// TIA Portal V17 export
// export: Created 2025-03-10T13:11:52.9134502Z, ExportSetting WithDefaults, DisplayName Totally Integrated Automation Portal, DisplayVersion V17 Update 8, DisplayName TIA Portal Openness, DisplayVersion V17 Update 8, DisplayName TIA Portal Version Control Interface, DisplayVersion V17, DisplayName SINAMICS Startdrive Advanced, DisplayVersion V17 SP2, DisplayName SINAMICS Startdrive G110M, G120, G120C, G120D, G120P, G115D, DisplayVersion V17 SP2, DisplayName SINAMICS Startdrive G130, G150, S120, S150, SINAMICS MV, S210, DisplayVersion V17 SP2, DisplayName STEP 7 Professional, DisplayVersion V17 Update 8, DisplayName SINUMERIK ONE STEP 7 Toolbox, DisplayVersion V17 Update 12, DisplayName SINUMERIK 840D sl STEP 7 Toolbox, DisplayVersion V17 Update 12, DisplayName STEP 7 Safety, DisplayVersion V17 Update 6, DisplayName WinCC Advanced, DisplayVersion V17 Update 8
TYPE "LBP_typeChanX"
TITLE = Channel interface / Interfaz de canal / Kanalschnittstelle
// User data type for blocks LBP_Chan1 [DB21] .. LBP_Chan10 [DB30] / Tipo de dato de usuario para bloques LBP_Chan1 [DB21] .. LBP_Chan10 [DB30] / Anwender-Datentyp für Bausteine LBP_Chan1 [DB21] .. LBP_Chan10 [DB30]
// stored: IsFailsafeCompliant false
   STRUCT
      f0_0 : Bool;
      f0_1 : Bool;
      f0_2 : Bool;
      A_DRF : Bool;   // DRF aktivieren / Activate DRF / Activar DRF
      A_SBL : Bool;   // Einzelsatz aktivieren / Activate single block / Activar secuencia individual
      A_M01 : Bool;   // M01 aktivieren / Activate M01 / Activar M01
      A_DRY : Bool;   // Probelauf Vorschub aktivieren / Activate dry run feedrate / Activar avance recorrido de prueba
      f0_7 : Bool;
      A_Ref : Bool;   // Referenzieren aktivieren / Activate referencing / Activar referenciado
      A_ProtZone : Bool;   // Schutzbereiche aktivieren / Enable protection zones / Activar zonas protegidas
      A_SynOff : Bool;   // Synchronaktion Aus / Synchronous action off / Acción síncrona desactivada
      A_TM_TimOut : Bool;   // Timeout aktivieren (TM) / Activate time-out (TM) / Activar timeout (TM)
      A_CLC_Stop : Bool;   // CLC Stopp / CLC stop / Parada CLC
      A_CLC_OR : Bool;   // CLC Override / CLC override / Corrección CLC
      A_PLC_ActCompl : Bool;   // PLC-Aktion abgeschlossen / PLC action completed / Acción PLC finalizada
      A_ProgTest : Bool;   // Programmtest aktivieren / Activate program test / Activar test de programa
      A_SKP0 : Bool;   // Ausblendsatz \0 aktivieren / Activate skip block \0 / Activar omisión de bloque \0
      A_SKP1 : Bool;   // Ausblendsatz \1 aktivieren / Activate skip block \1 / Activar omisión de bloque \1
      A_SKP2 : Bool;   // Ausblendsatz \2 aktivieren / Activate skip block \2 / Activar omisión de bloque \2
      A_SKP3 : Bool;   // Ausblendsatz \3 aktivieren / Activate skip block \3 / Activar omisión de bloque \3
      A_SKP4 : Bool;   // Ausblendsatz \4 aktivieren / Activate skip block \4 / Activar omisión de bloque \4
      A_SKP5 : Bool;   // Ausblendsatz \5 aktivieren / Activate skip block \5 / Activar omisión de bloque \5
      A_SKP6 : Bool;   // Ausblendsatz \6 aktivieren / Activate skip block \6 / Activar omisión de bloque \6
      A_SKP7 : Bool;   // Ausblendsatz \7 aktivieren / Activate skip block \7 / Activar omisión de bloque \7
      A_StrokEnab : Bool;   // Hub aktivieren / Stroke enable / Activar carrera
      A_ManStrokEnab : Bool;   // Manuelle Hub-Aktivierung / Manual stroke enable / Habilitación manual de carrera
      A_StrokSup : Bool;   // Hub-Unterdrückung / Stroke suppression / Supresión de carrera
      A_StrokDelayed : Bool;   // Hub verzögert / Stroke delayed / Carrera retardada
      A_StrokStop : Bool;   // Hub läuft nicht / Stroke not operating / Carrera no en ejecución
      A_ManRelStroke2 : Bool;   // Manuelle Freigabe von Hub 2 / Manual release of stroke 2 / Habilitación manual de carrera 2
      A3_6 : Bool;
      A3_7 : Bool;
      A_FD_OR : Byte;   // Vorschub-Override / Feedrate override / Corrección de avance
      A_RT_OR : Byte;   // Eilgang Override / Rapid traverse override / Corregir rápido
      A_FDdisable : Bool;   // Vorschub deaktivieren / Feed disable / Desactivar avance
      A_RIdisable : Bool;   // Einlesen deaktivieren / Read-in disable / Desactivar lectura
      A_DeleteDTG : Bool;   // Restweg löschen / Delete distance to go / Borrar trayecto residual
      A_SP_Clear : Bool;   // UP Anzahl der Arbeitsgänge löschen / Delete UP number of passes / Borrar número UP de operaciones
      A_ProgAbort : Bool;   // Abbruch Programmebene / Program level abort / Cancelar nivel de programa
      A_F_Limit : Bool;   // Werkzeugbahn Vorschub-Begrenzung / Tool path feedrate limitation / Limitación avance trayecto de herramienta
      A_RT_ORA : Bool;   // Eilgang Override aktiv / Rapid traverse override active / Corrección rápido activa
      A_FD_ORA : Bool;   // Vorschub Override aktiv / Feedrate override active / Corrección avance activa
      A_NCStartDisabl : Bool;   // NC Start deaktivieren / NC start disable / Desactivar Marcha CN
      A_NCStart : Bool;   // NC Start / NC start / Marcha CN
      A_NCStopBlock : Bool;   // NC Stopp an Satzgrenze / NC stop at block limit / Parada CN en límite de bloque
      A_NCStop : Bool;   // NC Stopp / NC stop / Parada CN
      A_NCStopASp : Bool;   // NC Stopp-Achsen plus Spindel / NC stop axes plus spindle / Parada CN ejes y cabezal
      A_SuppStartLock : Bool;   // Startsperre unterdrücken / Suppress Start Lock / Suprimir bloqueo de arranque
      A_CfgStopFunc : Bool;   // Konfigurierte Stopp-Funktion aktivieren / Activate configured stop function / Activar la función de parada configurada
      A_Reset : Bool;   // Reset
      A_MRP : Array[1..10] of Bool;   // Maschinenbezogenen Schutzbereich aktivieren [1..10] / Activate machine-related protection zone [1..10] / Activar zona protegida específica de máquina [1..10]
      A_CSP : Array[1..10] of Bool;   // Kanalspezifische Schutzbereich aktivieren [1..10] / Activate channel-specific protection zone [1..10] / Activar zona protegida específica de canal [1..10]
      A_Geo : Array[1..3] of Struct   // Steuersignale für Geometrieachse [1..3] / Control signals for geometry axis [1..3] / Señales de control para eje geométrico [1..3]
         HW1 : Bool;   // Handrad 1 aktivieren / Activate handwheel 1 / Activar volante 1
         HW2 : Bool;   // Handrad 2 aktivieren / Activate handwheel 2 / Activar volante 2
         HW3 : Bool;   // Handrad 3 aktivieren / Activate handwheel 3 / Activar volante 3
         FDStop : Bool;   // Vorschub Stopp / Feedrate stop / Parada de avance
         Disabl : Bool;   // Verfahrtaste deaktivieren / Traversing key disable / Desactivar tecla de desplazamiento
         RapidTrOR : Bool;   // Eilgang Override / Rapid traverse override / Corregir rápido
         Minus : Bool;   // Verfahrtaste minus / Traversing key minus / Tecla desplazamiento Menos
         Plus : Bool;   // Verfahrtaste plus / Traversing key plus / Tecla desplazamiento Más
         INC1 : Bool;   // INC 1
         INC10 : Bool;   // INC 10
         INC100 : Bool;   // INC 100
         INC1000 : Bool;   // INC 1000
         INC10000 : Bool;   // INC 10000
         INCVar : Bool;   // INC-Variable / INC variable / Variable INC
         ContManTravel : Bool;   // Kontinuierliches Verfahren von Hand / Continuous manual travel / Desplazamiento continuo a mano
         f1_7 : Bool;
         OEM : Byte;   // OEM-Signale / OEM signals / Señales OEM
         InvHWDirOfRot : Bool;   // Handrad-Drehrichtung umkehren / Invert handwheel direction of rotation / Invertir sentido de giro de volante
         f3_1 : Bool;
         f3_2 : Bool;
         f3_3 : Bool;
         f3_4 : Bool;
         f3_5 : Bool;
         f3_6 : Bool;
         f3_7 : Bool;
      END_STRUCT;
      f24_0 : Bool;
      E_MMC_CfgStopFunc : Bool;   // HMI: Konfigurierte Stopp-Funktion (CST) ist angewählt / HMI: configured stop function (CST) is selected / HMI: La función de parada configurada (CST) está seleccionada
      f24_2 : Bool;
      E_MMC_DRF : Bool;   // HMI DRF ausgewählt / HMI DRF selected / HMI DRF seleccionado
      E_MMC_M01AssocNC : Bool;   // M01 verbunden mit NC auswählen / Select M01 associated with NC / Seleccionar M01 asociado a CN
      E_MMC_M01 : Bool;   // HMI M01 ausgewählt / HMI M01 selected / HMI M01 seleccionado
      E_MMC_DRY : Bool;   // HMI Probelauf Vorschub ausgewählt / HMI Dry-run feedrate selected / HMI Recorrido de prueba avance seleccionado
      f24_7 : Bool;
      E_MMC_REPOSPM_0 : Bool;   // HMI REPOSPATHMODE 0
      E_MMC_REPOSPM_1 : Bool;   // HMI REPOSPATHMODE 1
      E_MMC_REPOSPM_2 : Bool;   // HMI REPOSPATHMODE 2
      E_MMC_FD_OR4RT_OR : Bool;   // HMI Vorschub Override für Eilgang ausgewählt / HMI Feedrate override for rapid traverse selected / HMI Corrección avance para rápido seleccionada
      E_MMC_REPOSMode : Bool;   // HMI REPOS MODE EDGE
      f25_5 : Bool;
      f25_6 : Bool;
      E_MMC_ProgTest : Bool;   // Programmtest ausgewählt / Program test selected / Test de programa seleccionado
      E_MMC_SKP0 : Bool;   // HMI-Baustein überspringen ausgewählt \0 / HMI skip block selected \0 / Omitir bloque HMI seleccionado \0
      E_MMC_SKP1 : Bool;   // HMI-Baustein überspringen ausgewählt \1 / HMI skip block selected \1 / Omitir bloque HMI seleccionado \1
      E_MMC_SKP2 : Bool;   // HMI-Baustein überspringen ausgewählt \2 / HMI skip block selected \2 / Omitir bloque HMI seleccionado \2
      E_MMC_SKP3 : Bool;   // HMI-Baustein überspringen ausgewählt \3 / HMI skip block selected \3 / Omitir bloque HMI seleccionado \3
      E_MMC_SKP4 : Bool;   // HMI-Baustein überspringen ausgewählt \4 / HMI skip block selected \4 / Omitir bloque HMI seleccionado \4
      E_MMC_SKP5 : Bool;   // HMI-Baustein überspringen ausgewählt \5 / HMI skip block selected \5 / Omitir bloque HMI seleccionado \5
      E_MMC_SKP6 : Bool;   // HMI-Baustein überspringen ausgewählt \6 / HMI skip block selected \6 / Omitir bloque HMI seleccionado \6
      E_MMC_SKP7 : Bool;   // HMI-Baustein überspringen ausgewählt \7 / HMI skip block selected \7 / Omitir bloque HMI seleccionado \7
      E_MMC_SKP8 : Bool;   // HMI-Baustein überspringen ausgewählt \8 / HMI skip block selected \8 / Omitir bloque HMI seleccionado \8
      E_MMC_SKP9 : Bool;   // HMI-Baustein überspringen ausgewählt \9 / HMI skip block selected \9 / Omitir bloque HMI seleccionado \9
      f27_2 : Bool;
      f27_3 : Bool;
      f27_4 : Bool;
      f27_5 : Bool;
      f27_6 : Bool;
      f27_7 : Bool;
      A_OEM : Byte;
      A_FixedFD1 : Bool;   // Festen Vorschub 1 aktivieren / Activate fixed feedrate 1 / Activar avance fijo 1
      A_FixedFD2 : Bool;   // Festen Vorschub 2 aktivieren / Activate fixed feedrate 2 / Activar avance fijo 2
      A_FixedFD3 : Bool;   // Festen Vorschub 3 aktivieren / Activate fixed feedrate 3 / Activar avance fijo 3
      A_FixedFD4 : Bool;   // Festen Vorschub 4 aktivieren / Activate fixed feedrate 4 / Activar avance fijo 4
      A_PTP_Travel : Bool;   // PTP Verfahren aktivieren / Activate PTP traversal / Activar desplazamiento PTP
      A_DisablWP_Counter : Bool;   // Werkstückzähler deaktivieren / Deactivate workpiece counter / Desactivar contador de piezas
      A_DisablWearMon : Bool;   // Verschleißüberwachung deaktivieren / Deactivate wear monitoring / Desactivar vigilancia de desgaste
      A_DontDisablTool : Bool;   // Werkzeug nicht deaktivieren / Do not disable tool / No desactivar herramienta
      A_ContHW1 : Bool;   // Kontur-Handrad 1 aktivieren / Activate contour handwheel 1 / Activar volante de contorno 1
      A_ContHW2 : Bool;   // Kontur-Handrad 2 aktivieren / Activate contour handwheel 2 / Activar volante de contorno 2
      A_ContHW3 : Bool;   // Kontur-Handrad 3 aktivieren / Activate contour handwheel 3 / Activar volante de contorno 3
      A_ContHWsim : Bool;   // Simuliertes Kontur-Handrad Ein / Simulated contour handwheel on / Volante de contorno simulado Con
      A_ContHWneg : Bool;   // Kontur-Handrad neg. Weg / Contour handwheel neg. route / Volante de contorno trayecto neg.
      A_NCKrelatedM01 : Bool;   // NCK-bezogenes M01 aktivieren / Activate NCK-related M01 / Activar M01 referido al NCK
      A_JOG_Circles : Bool;   // JOG in Kreisen / JOG in circles / JOG en círculos
      A_NoToolChangeCmd : Bool;   // Keine Werkzeugwechselbefehle / No tool change commands / Sin comandos de cambio de herramientas
      A_REPOSPM_0 : Bool;   // REPOSPATHMODE 0
      A_REPOSPM_1 : Bool;   // REPOSPATHMODE 1
      A_REPOSPM_2 : Bool;   // REPOSPATHMODE 2
      f31_3 : Bool;
      A_REPOSMode : Bool;   // REPOS MODE EDGE
      A_InvCHWDirOfRot : Bool;   // Kontur-Handrad-Drehrichtung wird umgekehrt / Inverting contour handwheel direction of rotation / Se invierte en sentido de giro del volante de contorno
      A_SKP8 : Bool;   // Ausblendsatz \8 aktivieren / Activate skip block \8 / Activar omisión de bloque \8
      A_SKP9 : Bool;   // Ausblendsatz \9 aktivieren / Activate skip block \9 / Activar omisión de bloque \9
      E_ExecExtern : Bool;   // Ausführung aus externer Quelle aktiv / Execution from external source active / Ejecución desde fuente externa activa
      f32_1 : Bool;
      f32_2 : Bool;
      E_ActBlock : Bool;   // Aktionsbaustein aktiv / Action block active / Bloque de acción activo
      E_BegBlock : Bool;   // Anfahrsatz aktiv / Approach block active / Secuencia de aproximación activo
      E_M01 : Bool;   // M0/M1 aktiv / M0/M1 active / M0/M1 activo
      E_LastActBlock : Bool;   // Letzter Aktionsbaustein aktiv / Last action block active / Último bloque de acción activo
      f32_7 : Bool;
      E_Ref : Bool;   // Referenzieren aktiv / Referencing active / Referenciado activo
      E_OrieToolholder : Bool;   // Orientierbarer Werkzeughalter aktiv / Orientable toolholder active / Portaherramientas orientable activo
      E_RevFD : Bool;   // Umdrehungsvorschub aktiv / Revolutional feedrate active / Avance revoluciones activo
      E_HWOverlay : Bool;   // Handrad Override aktiv / Handwheel override active / Corrección volante activa
      E_BlockSearch : Bool;   // Satzsuche aktiv / Block search active / Búsqueda de secuencia activa
      E_M30 : Bool;   // M2/M30 aktiv / M2/M30 active / M2/M30 activo
      E_Transform : Bool;   // Transformation aktiv / Transformation active / Transformación activa
      E_ProgTest : Bool;   // Programmtest aktiv / Program test active / Test de programa activo
      E_OEMChan : Byte;   // Rückmeldung OEM Kanalsignale / OEM channel signals feedback / Respuesta OEM señales de canal
      E_ProgRunning : Bool;   // Programm läuft / Program running / Programa en ejecución
      E_ProgWait : Bool;   // Programm wartet / Program waiting / Programa en espera
      E_ProgStop : Bool;   // Programm gestoppt / Program stopped / Programa detenido
      E_ProgInterrupt : Bool;   // Programm unterbrochen / Program interrupted / Programa interrumpido
      E_ProgAborted : Bool;   // Programm abgebrochen / Program aborted / Programa cancelado
      E_ChanActive : Bool;   // Kanal aktiv / Channel active / Canal activo
      E_ChanInterrupt : Bool;   // Kanal unterbrochen / Channel interrupted / Canal interrumpido
      E_ChanReset : Bool;   // Kanal Reset / Channel reset / Reset de canal
      E_StartReq : Bool;   // Startanforderung / Start request / Solicitud arranque
      E_StopReq : Bool;   // Stoppanforderung / Stop request / Solicitud parada
      E_AxesRef : Bool;   // Alle Achsen referenziert / All axes referenced / Todos los ejes referenciados
      E_AxesStop : Bool;   // Alle Achsen im Stillstand / All axes stationary / Todos los ejes en parada
      E_IR_Activ : Bool;   // Interruptverarbeitung aktiv / Interrupt processing active / Tratamiento de interrupciones activo
      E_ChanRO : Bool;   // Kanal betriebsbereit / Channel ready for operation / Canal listo para funcionar
      E_NCKalarmChan : Bool;   // Kanalspezifischer NCK-Alarm steht an / Channel-specific NCK alarm present / Alarma de NCK específica de canal presente
      E_NCKalarmStop : Bool;   // NCK-Alarm mit Bearbeitungsstopp steht an / NCK alarm with processing stop present / Alarma de NCK con parada del mecanizado presente
      E_CHW1 : Bool;   // Kontur-Handrad 1 Ein / Contour handwheel 1 on / Volante de contorno 1 Con
      E_CHW2 : Bool;   // Kontur-Handrad 2 Ein / Contour handwheel 2 on / Volante de contorno 2 Con
      E_CHW3 : Bool;   // Kontur-Handrad 3 Ein / Contour handwheel 3 on / Volante de contorno 3 Con
      E_CLC : Bool;   // CLC aktiv / CLC active / CLC activo
      E_CLCStopLL : Bool;   // CLC gestoppt Untergrenze / CLC stopped lower limit / CLC detenido límite inferior
      E_CLCStopUL : Bool;   // CLC gestoppt Obergrenze / CLC stopped upper limit / CLC detenido límite superior
      E_RIEnabIgnored : Bool;   // Aktivierung Einlesen wird ignoriert / Read-in enable is ignored / Activación de lectura se ignora
      E_StopBlkEndSBLsuppr : Bool;   // Stopp am Satzende bei SBL unterdrückt / Stop at block end with SBL is suppressed / Parada en final de secuencia con SBL suprimido
      E_StrokeEA : Bool;   // Hubfreigabe aktiv / Stroke release active / Habilitación de carrera activa
      E_AcknManStrokEnab : Bool;   // Quittierung manuelle Hubfreigabe / Acknowledgment of manual stroke release / Confirmación habilitación manual de carrera
      f38_2 : Bool;
      f38_3 : Bool;
      f38_4 : Bool;
      f38_5 : Bool;
      f38_6 : Bool;
      f38_7 : Bool;
      E_ProtZoneNOK : Bool;   // Schutzbereiche nicht garantiert / Protection zones not guaranteed / Zonas protegidas no garantizadas
      E_NCalarmWithProgStop : Bool;   // NC-Alarm mit Programmstopp / NC alarm with program stop / Alarma de CN con parada de programa
      f39_2 : Bool;
      f39_3 : Bool;
      E_SblStopAtBlockEnd : Bool;   // Stopp am Satzende aufgrund des Einzelsatzes / Stop at block end due to single block / Parada en final de secuencia debido a la secuencia individual
      E_InvCHWDirOfRot : Bool;   // Aktive Umkehr der Kontur-Handrad-Drehrichtung / Contour handwheel direction of rotation invert actively / Inversión activa del sentido de giro volante de contorno
      E_CfgStopFuncActive : Bool;   // Konfigurierte Stopp-Funktion ist aktiviert / Configured stop function is activated / La función de parada configurada está activada
      E_CfgStopAtBlockEnd : Bool;   // Stopp am Satzende aufgrund des konfigurierten Stopps / Stop at block end due to configured stop / Parada en final de secuencia debido a la parada configurada
      E_Geo : Array[1..3] of Struct   // Statussignale der Geometrieachse [1..3] / Status signals of geometry axis [1..3] / Señales de estado del eje geométrico [1..3]
         HW1 : Bool;   // Handrad 1 aktiv / Handwheel 1 active / Volante 1 activo
         HW2 : Bool;   // Handrad 2 aktiv / Handwheel 2 active / Volante 2 activo
         HW3 : Bool;   // Handrad 3 aktiv / Handwheel 3 active / Volante 3 activo
         f0_3 : Bool;
         TReqMinus : Bool;   // Verfahranforderungen minus / Travel requests minus / Solicitudes de desplazamiento Menos
         TReqPlus : Bool;   // Verfahranforderungen plus / Travel requests plus / Solicitudes de desplazamiento Más
         TCMinus : Bool;   // Verfahrbefehl minus / Traverse command minus / Comando de desplazamiento Menos
         TCPlus : Bool;   // Verfahrbefehl plus / Traverse command plus / Comando de desplazamiento Más
         INC1 : Bool;   // INC 1 aktiv / INC 1 active / INC 1 activo
         INC10 : Bool;   // INC 10 aktiv / INC 10 active / INC 10 activo
         INC100 : Bool;   // INC 100 aktiv / INC 100 active / INC 100 activo
         INC1000 : Bool;   // INC 1000 aktiv / INC 1000 active / INC 1000 activo
         INC10000 : Bool;   // INC 10000 aktiv / INC 10000 active / INC 10000 activo
         INCVar : Bool;   // INC-Variable aktiv / INC variable active / Variable INC activa
         ContManTravelAct : Bool;   // Kontinuierliches manuelles Verfahren aktiv / Continuous manual travel active / Desplazamiento manual continuo activo
         f1_7 : Bool;
         OEM : Byte;   // OEM-Signale / OEM signals / Señales OEM
         InvHWDirOfRot : Bool;   // Handrad-Drehrichtung invertiert aktiv / Handwheel direction of rotation invert actively / Invertir activamente sentido de giro volante
         f3_1 : Bool;
         f3_2 : Bool;
         f3_3 : Bool;
         f3_4 : Bool;
         f3_5 : Bool;
         f3_6 : Bool;
         f3_7 : Bool;
         f4 : Byte;
      END_STRUCT;
      M1Change : Bool;   // M-Funktion 1 Änderung / M function 1 change / Modificación función M 1
      M2Change : Bool;   // M-Funktion 2 Änderung / M function 2 change / Modificación función M 2
      M3Change : Bool;   // M-Funktion 3 Änderung / M function 3 change / Modificación función M 3
      M4Change : Bool;   // M-Funktion 4 Änderung / M function 4 change / Modificación función M 4
      M5Change : Bool;   // M-Funktion 5 Änderung / M function 5 change / Modificación función M 5
      f58_5 : Bool;
      f58_6 : Bool;
      f58_7 : Bool;
      M1NDec : Bool;   // M-Funktion 1 nicht decodiert / M function 1 not decoded / Función M 1 no decodificada
      M2NDec : Bool;   // M-Funktion 2 nicht decodiert / M function 2 not decoded / Función M 2 no decodificada
      M3NDec : Bool;   // M-Funktion 3 nicht decodiert / M function 3 not decoded / Función M 3 no decodificada
      M4NDec : Bool;   // M-Funktion 4 nicht decodiert / M function 4 not decoded / Función M 4 no decodificada
      M5NDec : Bool;   // M-Funktion 5 nicht decodiert / M function 5 not decoded / Función M 5 no decodificada
      f59_5 : Bool;
      f59_6 : Bool;
      f59_7 : Bool;
      S1Change : Bool;   // S-Funktion 1 Änderung / S function 1 change / Modificación función S 1
      S2Change : Bool;   // S-Funktion 2 Änderung / S function 2 change / Modificación función S 2
      S3Change : Bool;   // S-Funktion 3 Änderung / S function 3 change / Modificación función S 3
      f60_3 : Bool;
      S1Quick : Bool;   // S-Funktion 1 schnell / S function 1 quick / Función S 1 rápida
      S2Quick : Bool;   // S-Funktion 2 schnell / S function 2 quick / Función S 2 rápida
      S3Quick : Bool;   // S-Funktion 3 schnell / S function 3 quick / Función S 3 rápida
      f60_7 : Bool;
      T1Change : Bool;   // T-Funktion 1 Änderung / T function 1 change / Modificación función T 1
      T2Change : Bool;   // T-Funktion 2 Änderung / T function 2 change / Modificación función T 2
      T3Change : Bool;   // T-Funktion 3 Änderung / T function 3 change / Modificación función T 3
      f61_3 : Bool;
      T1Quick : Bool;   // T-Funktion 1 schnell / T function 1 quick / Función T 1 rápida
      T2Quick : Bool;   // T-Funktion 2 schnell / T function 2 quick / Función T 2 rápida
      T3Quick : Bool;   // T-Funktion 3 schnell / T function 3 quick / Función T 3 rápida
      f61_7 : Bool;
      D1Change : Bool;   // D-Funktion 1 Änderung / D function 1 change / Modificación función D 1
      D2Change : Bool;   // D-Funktion 2 Änderung / D function 2 change / Modificación función D 2
      D3Change : Bool;   // D-Funktion 3 Änderung / D function 3 change / Modificación función D 3
      f62_3 : Bool;
      D1Quick : Bool;   // D-Funktion 1 schnell / D function 1 quick / Función D 1 rápida
      D2Quick : Bool;   // D-Funktion 2 schnell / D function 2 quick / Función D 2 rápida
      D3Quick : Bool;   // D-Funktion 3 schnell / D function 3 quick / Función D 3 rápida
      f62_7 : Bool;
      EChange : Bool;   // E-Funktion Änderung / E function change / Modificación función E
      f63_1 : Bool;
      f63_2 : Bool;
      f63_3 : Bool;
      EQuick : Bool;   // E-Funktion schnell / E function quick / Función E rápida
      f63_5 : Bool;
      f63_6 : Bool;
      f63_7 : Bool;
      H1Change : Bool;   // H-Funktion 1 Änderung / H function 1 change / Modificación función H 1
      H2Change : Bool;   // H-Funktion 2 Änderung / H function 2 change / Modificación función H 2
      H3Change : Bool;   // H-Funktion 3 Änderung / H function 3 change / Modificación función H 3
      f64_3 : Bool;
      H1Quick : Bool;   // H-Funktion 1 schnell / H function 1 quick / Función H 1 rápida
      H2Quick : Bool;   // H-Funktion 2 schnell / H function 2 quick / Función H 2 rápida
      H3Quick : Bool;   // H-Funktion 3 schnell / H function 3 quick / Función H 3 rápida
      f64_7 : Bool;
      F1Change : Bool;   // F-Funktion 1 Änderung / F function 1 change / Modificación función F 1
      F2Change : Bool;   // F-Funktion 2 Änderung / F function 2 change / Modificación función F 2
      F3Change : Bool;   // F-Funktion 3 Änderung / F function 3 change / Modificación función F 3
      F4Change : Bool;   // F-Funktion 4 Änderung / F function 4 change / Modificación función F 4
      F5Change : Bool;   // F-Funktion 5 Änderung / F function 5 change / Modificación función F 5
      F6Change : Bool;   // F-Funktion 6 Änderung / F function 6 change / Modificación función F 6
      f65_6 : Bool;
      f65_7 : Bool;
      M1Quick : Bool;   // M-Funktion 1 schnell / M function 1 quick / Función M 1 rápida
      M2Quick : Bool;   // M-Funktion 2 schnell / M function 2 quick / Función M 2 rápida
      M3Quick : Bool;   // M-Funktion 3 schnell / M function 3 quick / Función M 3 rápida
      M4Quick : Bool;   // M-Funktion 4 schnell / M function 4 quick / Función M 4 rápida
      M5Quick : Bool;   // M-Funktion 5 schnell / M function 5 quick / Función M 5 rápida
      f66_5 : Bool;
      f66_6 : Bool;
      f66_7 : Bool;
      F1Quick : Bool;   // F-Funktion 1 schnell / F function 1 quick / Función F 1 rápida
      F2Quick : Bool;   // F-Funktion 2 schnell / F function 2 quick / Función F 2 rápida
      F3Quick : Bool;   // F-Funktion 3 schnell / F function 3 quick / Función F 3 rápida
      F4Quick : Bool;   // F-Funktion 4 schnell / F function 4 quick / Función F 4 rápida
      F5Quick : Bool;   // F-Funktion 5 schnell / F function 5 quick / Función F 5 rápida
      F6Quick : Bool;   // F-Funktion 6 schnell / F function 6 quick / Función F 6 rápida
      f67_6 : Bool;
      f67_7 : Bool;
      ExtM1 : Int;   // Erweiterte Adress-M-Funktion 1 (16 Bit INT) / Extended address M function 1 (16 bit INT) / Dirección ampliada función M 1 (16 bits INT)
      M1 : DInt;   // M-Funktion 1 (DInt) / M function 1 (DInt) / Función M 1 (DInt)
      ExtM2 : Int;   // Erweiterte Adress-M-Funktion 1 (16 Bit INT) / Extended address M function 1 (16 bit INT) / Dirección ampliada función M 1 (16 bits INT)
      M2 : DInt;   // M-Funktion 2 (DInt) / M function 2 (DInt) / Función M 2 (DInt)
      ExtM3 : Int;   // Erweiterte Adress-M-Funktion 1 (16 Bit INT) / Extended address M function 1 (16 bit INT) / Dirección ampliada función M 1 (16 bits INT)
      M3 : DInt;   // M-Funktion 3 (DInt) / M function 3 (DInt) / Función M 3 (DInt)
      ExtM4 : Int;   // Erweiterte Adress-M-Funktion 1 (16 Bit INT) / Extended address M function 1 (16 bit INT) / Dirección ampliada función M 1 (16 bits INT)
      M4 : DInt;   // M-Funktion 4 (DInt) / M function 4 (DInt) / Función M 4 (DInt)
      ExtM5 : Int;   // Erweiterte Adress-M-Funktion 1 (16 Bit INT) / Extended address M function 1 (16 bit INT) / Dirección ampliada función M 1 (16 bits INT)
      M5 : DInt;   // M-Funktion 5 (DInt) / M function 5 (DInt) / Función M 5 (DInt)
      ExtS1 : Int;   // Erweiterte Adress-S-Funktion 1 (16 Bit INT) / Extended address S function 1 (16 bit INT) / Dirección ampliada función S 1 (16 bits INT)
      S1 : Real;   // S-Funktion 1 (REAL) / S function 1 (REAL) / Función S 1 (REAL)
      ExtS2 : Int;   // Erweiterte Adress-S-Funktion 2 (16 Bit INT) / Extended address S function 2 (16 bit INT) / Dirección ampliada función S 2 (16 bits INT)
      S2 : Real;   // S-Funktion 2 (REAL) / S function 2 (REAL) / Función S 2 (REAL)
      ExtS3 : Int;   // Erweiterte Adress-S-Funktion 3 (16 Bit INT) / Extended address S function 3 (16 bit INT) / Dirección ampliada función S 3 (16 bits INT)
      S3 : Real;   // S-Funktion 3 (REAL) / S function 3 (REAL) / Función S 3 (REAL)
      ExtT1 : Int;   // Erweiterte Adress-T-Funktion 1 (16 Bit INT)T : DINT; //T-Funkton (DInt)f122 : INT;f124 : INT;f126 : INT; //Änderung falls 8-stellige T-Funktion / Extended address T function 1 (16 bit INT)T : DINT; //T function (DInt)f122 : INT;f124 : INT;f126 : INT; //Change in case of 8-digit T function / Dirección ampliada función T 1 (16 Bit INT)T : DINT; //Función T (DInt)f122 : INT;f124 : INT;f126 : INT; //Cambio en caso de función T de 8 dígitos
      T1 : Int;   // T-Funktion 1 (INT) / T function 1 (INT) / Función T 1 (INT)
      ExtT2 : Int;   // Erweiterte Adress-T-Funktion 2 (16 Bit INT) / Extended address T function 2 (16 bit INT) / Dirección ampliada función T 2 (16 bits INT)
      T2 : Int;   // T-Funktion 2 (INT) / T function 2 (INT) / Función T 2 (INT)
      ExtT3 : Int;   // Erweiterte Adress-T-Funktion 3 (16 Bit INT) / Extended address T function 3 (16 bit INT) / Dirección ampliada función T 3 (16 bits INT)
      T3 : Int;   // T-Funktion 3 (INT) / T function 3 (INT) / Función T 3 (INT)
      ExtD1 : Byte;   // Erweiterte Adress-D-Funktion 1 (8 Bit INT)D : INT;f132 : INT; //Änderung falls 5-stellige D-Funktion / Extended address D function 1 (8 bit INT)D : INT;f132 : INT; //Change in case of 5-digit D function / Dirección ampliada función D 1 (8 bits INT)D : INT;f132 : INT; //Cambio en caso de función de 5 dígitos
      D1 : Byte;   // D-Funktion 1 (8 Bit INT) / D function 1 (8 bit INT) / Función D 1 (8 bits INT)
      ExtD2 : Byte;   // Erweiterte Adress-D-Funktion 2 (8 Bit INT) / Extended address D function 2 (8 bit INT) / Dirección ampliada función D 2 (8 bits INT)
      D2 : Byte;   // D-Funktion 2 (8 Bit INT) / D function 2 (8 bit INT) / Función D 2 (8 bits INT)
      ExtD3 : Byte;   // Erweiterte Adress-D-Funktion 3 (8 Bit INT) / Extended address D function 3 (8 bit INT) / Dirección ampliada función D 3 (8 bits INT)
      D3 : Byte;   // D-Funktion 3 (8 Bit INT) / D function 3 (8 bit INT) / Función D 3 (8 bits INT)
      ExtE : Int;   // Erweiterte Adress-D-Funktion 3 (16 Bit INT) / Extended address D function 3 (16 bit INT) / Dirección ampliada función D 3 (16 bits INT)
      "E" : Real;   // E-Funktion (REAL) / E function (REAL) / Función E (REAL)
      ExtH1 : Int;   // Erweiterte Adress-H-Funktion 1 (16 Bit INT) / Extended address H function 1 (16 bit INT) / Dirección ampliada función H 1 (16 bits INT)
      H1 : Real;   // H-Funktion 1 (REAL), DInt auch in DBD396 / H function 1 (REAL), DInt also in DBD396 / Función H 1 (REAL), DInt también en DBD396
      ExtH2 : Int;   // Erweiterte Adress-H-Funktion 2 (16 Bit INT) / Extended address H function 2 (16 bit INT) / Dirección ampliada función H 2 (16 bits INT)
      H2 : Real;   // H-Funktion 2 (REAL), DInt auch in DBD400 / H function 2 (REAL), DInt also in DBD400 / Función H 2 (REAL), DInt también en DBD400
      ExtH3 : Int;   // Erweiterte Adress-H-Funktion 3 (16 Bit INT) / Extended address H function 3 (16 bit INT) / Dirección ampliada función H 3 (16 bits INT)
      H3 : Real;   // H-Funktion 3 (REAL), DInt auch in DBD404 / H function 3 (REAL), DInt also in DBD404 / Función H 3 (REAL), DInt también en DBD404
      ExtF1 : Int;   // Erweiterte Adress-F-Funktion1 (16 Bit INT) / Extended address F function 1 (16 bit INT) / Dirección ampliada función F 1 (16 bits INT)
      F1 : Real;   // F-Funktion 1 (REAL) / F function 1 (REAL) / Función F 1 (REAL)
      ExtF2 : Int;   // Erweiterte Adress-F-Funktion2 (16 Bit INT) / Extended address F function 2 (16 bit INT) / Dirección ampliada función F 2 (16 bits INT)
      F2 : Real;   // F-Funktion 2 (REAL) / F function 2 (REAL) / Función F 2 (REAL)
      ExtF3 : Int;   // Erweiterte Adress-F-Funktion3 (16 Bit INT) / Extended address F function 3 (16 bit INT) / Dirección ampliada función F 3 (16 bits INT)
      F3 : Real;   // F-Funktion 3 (REAL) / F function 3 (REAL) / Función F 3 (REAL)
      ExtF4 : Int;   // Erweiterte Adress-F-Funktion4 (16 Bit INT) / Extended address F function 4 (16 bit INT) / Dirección ampliada función F 4 (16 bits INT)
      F4 : Real;   // F-Funktion 4 (REAL) / F function 4 (REAL) / Función F 4 (REAL)
      ExtF5 : Int;   // Erweiterte Adress-F-Funktion5 (16 Bit INT) / Extended address F function 5 (16 bit INT) / Dirección ampliada función F 5 (16 bits INT)
      F5 : Real;   // F-Funktion 5 (REAL) / F function 5 (REAL) / Función F 5 (REAL)
      ExtF6 : Int;   // Erweiterte Adress-F-Funktion6 (16 Bit INT) / Extended address F function 6 (16 bit INT) / Dirección ampliada función F 6 (16 bits INT)
      F6 : Real;   // F-Funktion 6 (REAL) / F function 6 (REAL) / Función F 6 (REAL)
      MDyn : Array[0..99] of Bool;   // Dynamische M-Funktionen [0..99] / Dynamic M functions [0..99] / Funciones M dinámicas [0..99]
      GAct : Array[1..64] of Byte;   // Aktive G-Funktion von Gruppe [1..64] / Active G function of group [1..64] / Función G activa del grupo [1..64]
      E_MRPactivated : Array[1..10] of Bool;   // Maschinenbezogener Schutzbereich [1..10] vorab aktiviert / Machine-related protection zone [1..10] preactivated / Zona protegida específica de máquina [1..10] activada previamente
      E_CSPactivated : Array[1..10] of Bool;   // Kanalspezifischer Schutzbereich [1..10] vorab aktiviert / Channel-specific protection zone [1..10] preactivated / Zona protegida específica de canal [1..10] preactivada
      E_MRPViolated : Array[1..10] of Bool;   // Maschinenbezogener Schutzbereich 1..10] verletzt / Machine-related protection zone [1..10] violated / Zona protegida específica de máquina [1..10] vulnerada
      E_CSPViolated : Array[1..10] of Bool;   // Kanalspezifischer Schutzbereich [1..10] verletzt ab P4 / Channel-specific protection zone [1..10] violated from P4 on / Zona protegida específica de canal [1..10] vulnerada a partir de P4
      f_280_0 : Bool;
      A_Str_Synon : Bool;   // Anforderung Synchronaktionen sperren / Request of syn.action to NCK / Solicitar acción síncrona al NCK
      f_280_2 : Bool;
      f_280_3 : Bool;
      f_280_4 : Bool;
      f_280_5 : Bool;
      f_280_6 : Bool;
      f_280_7 : Bool;
      f_281_0 : Bool;
      A_Str_Synfrom : Bool;   // Quittung Synchronaktionen gesperrt / Request syn.action from NCK / Solicitar acción síncrona desde NCK
      f_281_2 : Bool;
      f_281_3 : Bool;
      f_281_4 : Bool;
      f_281_5 : Bool;
      f_281_6 : Bool;
      f_281_7 : Bool;
      f_282 : Int;
      f_284 : Int;
      f_286 : Int;
      f_288 : Int;
      f_290 : Int;
      f_292 : Int;
      f_294 : Int;
      f_296 : Int;
      f_298 : Int;
      A_SynDisabl : Array[1..64] of Bool;   // Synchronaktionen deaktivieren / Disable synchronous actions / Deshabilitar acciones síncronas
      E_SynDisabled : Array[1..64] of Bool;   // Synchronaktionen deaktiviert / Synchronous actions disabled / Sincronización desactivada
      E_G00 : Bool;   // Aktive G-Funktionen / Active G functions / Funciones G activas
      f316_1 : Bool;
      f316_2 : Bool;
      f316_3 : Bool;
      f316_4 : Bool;
      f316_5 : Bool;
      f316_6 : Bool;
      f316_7 : Bool;
      E_ExtLang : Bool;   // Externer Sprachmodus aktiv / External language mode active / Modo de lenguaje externo activo
      E_WS_Setp : Bool;   // Werkstück-Sollwert erreicht / Workpiece setpoint reached / Consigna de pieza alcanzada
      f317_2 : Bool;
      f317_3 : Bool;
      f317_4 : Bool;
      E_DriveTest : Bool;   // Verfahranforderung Antriebstest / Travel request drive test / Solicitud desplazamiento prueba de accionamiento
      E_PTP_Travel : Bool;   // PTP Verfahren aktiv / PTP travel active / Desplazamiento PTP activo
      E_ToolMissing : Bool;   // Werkzeug fehlt / Tool missing / Falta herramienta
      E_ASUP_Stop : Bool;   // ASUP gestoppt / ASUP stopped / ASUP detenido
      E_SearchAct : Bool;   // Suche aktiv / Search active / Búsqueda activa
      E_TOFF : Bool;   // TOFF aktiv / TOFF active / TOFF activo
      E_TOFFmovem : Bool;   // TOFF Bewegung aktiv / TOFF motion active / Movimiento TOFF activo
      E_StopDelayed : Bool;   // Stopp verzögert / Stop delayed / Parada retardada
      E_AssM01 : Bool;   // Zugehöriges M01 aktiv / Associated M01 active / M01 asociado activo
      E_DRY : Bool;   // Probelauf Vorschub aktiv / Dry-run feedrate active / Recorrido de prueba avance activo
      E_Overstore : Bool;   // Overstore aktiv / Overstore active / Sobrememorización activa
      E_REPOS_EdgeAckn : Bool;   // REPOS MODE EDGE ACKN
      E_REPOS_PMode0 : Bool;   // REPOS Path Mode Ackn 0
      E_REPOS_PMode1 : Bool;   // REPOS Path Mode Ackn 1
      E_REPOS_PMode2 : Bool;   // REPOS Path Mode Ackn 2
      E_DelayFTS : Bool;   // Verzögerung FTS / Delay FTS / Retardo FTS
      E_REPOS_DEFERRA : Bool;   // REPOS DEFERRA L Chan
      E_Stop_NoDelayR : Bool;   // Stopp-Verzögerungsbereich nicht akzeptiert / Stop-delay area not accepted / Zona de retardo de parada no aceptada
      E_NoToolChangeCmd : Bool;   // Kein Werkzeugwechselbefehl aktiv / No tool change command active / No hay comando de cambio de herramienta activo
      A_Ori : Array[1..3] of Struct   // Steuersignale für Orientierungsachsen [1..3] / Control signals for orientation axes [1..3] / Señales de control para ejes de orientación [1..3]
         HW1 : Bool;   // Handrad 1 aktivieren / Activate handwheel 1 / Activar volante 1
         HW2 : Bool;   // Handrad 2 aktivieren / Activate handwheel 2 / Activar volante 2
         HW3 : Bool;   // Handrad 3 aktivieren / Activate handwheel 3 / Activar volante 3
         FDStop : Bool;   // Vorschub Stopp / Feedrate stop / Parada de avance
         Disabl : Bool;   // Verfahrtaste sperren / Traversing key lock / Bloquear tecla desplazamiento
         RapidTrOR : Bool;   // Eilgang Override / Rapid traverse override / Corregir rápido
         Minus : Bool;   // Verfahrtaste minus / Traversing key minus / Tecla desplazamiento Menos
         Plus : Bool;   // Verfahrtaste plus / Traversing key plus / Tecla desplazamiento Más
         INC1 : Bool;   // INC 1 aktiv / INC 1 active / INC 1 activo
         INC10 : Bool;   // INC 10 aktiv / INC 10 active / INC 10 activo
         INC100 : Bool;   // INC 100 aktiv / INC 100 active / INC 100 activo
         INC1000 : Bool;   // INC 1000 aktiv / INC 1000 active / INC 1000 activo
         INC10000 : Bool;   // INC 10000 aktiv / INC 10000 active / INC 10000 activo
         INCVar : Bool;   // INC-Variable aktiv / INC variable active / Variable INC activa
         OEM : Byte;   // OEM-Signale / OEM signals / Señales OEM
         InvHWDirOfRot : Bool;   // Drehrichtung Handrad umkehren / Inverting handwheel direction of rotation / Invertir sentido de giro volante
         f3_1 : Bool;
         f3_2 : Bool;
         f3_3 : Bool;
         f3_4 : Bool;
         f3_5 : Bool;
         f3_6 : Bool;
         f3_7 : Bool;
      END_STRUCT;
      E_Ori : Array[1..3] of Struct   // Steuersignale für Orientierungsachsen [1..3] / Control signals for orientation axes [1..3] / Señales de control para ejes de orientación [1..3]
         HW1 : Bool;   // Handrad 1 aktiv / Handwheel 1 active / Volante 1 activo
         HW2 : Bool;   // Handrad 2 aktiv / Handwheel 2 active / Volante 2 activo
         HW3 : Bool;   // Handrad 3 aktiv / Handwheel 3 active / Volante 3 activo
         f0_3 : Bool;
         TReqMinus : Bool;   // Verfahranforderungen minus / Travel requests minus / Solicitudes de desplazamiento Menos
         TReqPlus : Bool;   // Verfahranforderungen plus / Travel requests plus / Solicitudes de desplazamiento Más
         TCMinus : Bool;   // Verfahrbefehl minus / Traverse command minus / Comando de desplazamiento Menos
         TCPlus : Bool;   // Verfahrbefehl plus / Traverse command plus / Comando de desplazamiento Más
         INC1 : Bool;   // INC 1 aktiv / INC 1 active / INC 1 activo
         INC10 : Bool;   // INC 10 aktiv / INC 10 active / INC 10 activo
         INC100 : Bool;   // INC 100 aktiv / INC 100 active / INC 100 activo
         INC1000 : Bool;   // INC 1000 aktiv / INC 1000 active / INC 1000 activo
         INC10000 : Bool;   // INC 10000 aktiv / INC 10000 active / INC 10000 activo
         INCVar : Bool;   // INC-Variable aktiv / INC variable active / Variable INC activa
         OEM : Byte;   // OEM-Signale / OEM signals / Señales OEM
         InvHWDirOfRot : Bool;   // Handrad-Drehrichtung invertiert aktiv / Handwheel direction of rotation invert actively / Invertir activamente sentido de giro volante
         f3_1 : Bool;
         f3_2 : Bool;
         f3_3 : Bool;
         f3_4 : Bool;
         f3_5 : Bool;
         f3_6 : Bool;
         f3_7 : Bool;
      END_STRUCT;
      E_TPrewarnLimit : Bool;   // Werkzeug-Vorwarngrenze erreicht / Tool prewarn limit reached / Límite de prealarma alcanzado
      E_TLimit : Bool;   // Werkzeuggrenze erreicht / Tool limit reached / Límite de herramienta alcanzado
      E_TNewRepl : Bool;   // Übergang zu neuem Ersatzwerkzeug / Transition to new replacement tool / Transición a nueva herramienta de sustitución
      E_TLastRepl : Bool;   // Letztes Ersatzwerkzeug der Werkzeuggruppe / Last replacement tool of the tool group / Última herramienta de sustitución del grupo de herramientas
      f344_4 : Bool;
      f344_5 : Bool;
      f344_6 : Bool;
      f344_7 : Bool;
      f345 : Byte;
      f346 : Byte;
      f347 : Byte;
      E_TNoPrewarnLimit : DInt;   // WZ-Nummer für Werkzeug-Vorwarngrenze / T number for tool prewarn limit / Número de herramienta para límite de prealarma de herramienta
      E_TNoLimit : DInt;   // WZ-Nummer für Werkzeuggrenze / T number for tool limit / Número de herramienta para límite de herramienta
      E_TNoNewRepl : DInt;   // WZ-Nummer des neuen Ersatzwerkzeugs / T number of the new replacement tool / Número de herramienta de la nueva herramienta de sustitución
      E_TNoLastRepl : DInt;   // WZ-Nummer des letzten Ersatzwerkzeugs / T number of the last replacement tool / Número de herramienta de la última herramienta de sustitución
      E_Cycle_Sig : Array[0..15] of Bool;   // Zyklen-Eingangssignale / Cycles input signals / Señales de entrada de ciclos
      A_Cycle_Sig : Array[0..15] of Bool;   // Zyklen-Ausgangssignale / Cycles output signals / Señales de salida de ciclos
      E_OEM_TechnoSig : Array[0..31] of Bool;   // OEM Techno Eingangssignale / OEM Techno input signals / Señales de entrada OEM tecno
      A_OEM_TechnoSig : Array[0..31] of Bool;   // OEM Techno Ausgangssignale / OEM Techno output signals / Señales de salida OEM tecno
      E_ProgEvent_Start : Bool;   // Aktives Prog-Event: Start / Active Prog-Event: Start / Evento prog activo: arrancar
      E_ProgEvent_M30 : Bool;   // Aktives Prog-Event M30 / Active Prog-Event: M30 / Evento prog M30 activo
      E_ProgEvent_Reset : Bool;   // Aktives Prog-Event: Start / Active Prog-Event: Start / Evento prog activo: arrancar
      E_ProgEvent_PowerOn : Bool;   // Aktives Prog-Event: Einschalten / Active Prog-Event: Power on / Evento prog activo: encender
      E_ProgEvent_SearchRun : Bool;   // Aktives Prog-Event: Suche / Active Prog-Event: Search / Evento prog activo: buscar
      f376_5 : Bool;
      f376_6 : Bool;
      f376_7 : Bool;
      E_CollCheckStop : Bool;   // Stopp der Kollisionsprüfung / Stop of Collision Check / Parada de comprobación de colisiones
      E_StopCondition : Bool;   // Stoppbedingung / Stop Condition / Condición de parada
      f377_2 : Bool;
      f377_3 : Bool;
      E_JogRetract : Bool;   // JOG Rückzug aktiv / JOG Retract active / Retirada JOG activa
      E_RetractData : Bool;   // Rückzugsdaten verfügbar / Retract data available / Datos de retirada disponibles
      E_JOG_Circles : Bool;   // JOG in Kreisen / JOG in circles / JOG en círculos
      f377_7 : Bool;
      E_AnyAsup : Bool;   // AnyASUP aktiv / AnyASUP activ / AnyASUP activo
      E_SilentAsup : Bool;   // Stilles ASUP aktiv / Silent ASUP active / ASUP silencioso activo
      f378_2 : Bool;
      f378_3 : Bool;
      f378_4 : Bool;
      f378_5 : Bool;
      f378_6 : Bool;
      f378_7 : Bool;
      f379 : Byte;
      f380 : Array[0..31] of Bool;   // Reserviert / Reserved / Reservado
      A_ProgJump : Bool;   // Steuerprogramm Sprung / Control program jump / Salto programa de control
      f384_1 : Bool;
      f384_2 : Bool;
      f384_3 : Bool;
      f384_4 : Bool;
      f384_5 : Bool;
      f384_6 : Bool;
      f384_7 : Bool;
      A_InKeyG1 : Bool;   // Schleifsignal 1 / Grinding signal 1 / Señal de rectificado 1
      A_InKeyG2 : Bool;   // Schleifsignal 2 / Grinding signal 2 / Señal de rectificado 2
      A_InKeyG3 : Bool;   // Schleifsignal 3 / Grinding signal 3 / Señal de rectificado 3
      A_InKeyG4 : Bool;   // Schleifsignal 4 / Grinding signal 4 / Señal de rectificado 4
      A_InKeyG5 : Bool;   // Schleifsignal 5 / Grinding signal 5 / Señal de rectificado 5
      A_InKeyG6 : Bool;   // Schleifsignal 6 / Grinding signal 6 / Señal de rectificado 6
      A_InKeyG7 : Bool;   // Schleifsignal 7 / Grinding signal 7 / Señal de rectificado 7
      A_InKeyG8 : Bool;   // Schleifsignal 8 / Grinding signal 8 / Señal de rectificado 8
      A_InKeyGEn1 : Bool;   // Schleifsignal 1 aktivieren / Enable grinding signal 1 / Habilitar señal de rectificado 1
      A_InKeyGEn2 : Bool;   // Schleifsignal 2 aktivieren / Enable grinding signal 2 / Habilitar señal de rectificado 2
      A_InKeyGEn3 : Bool;   // Schleifsignal 3 aktivieren / Enable grinding signal 3 / Habilitar señal de rectificado 3
      A_InKeyGEn4 : Bool;   // Schleifsignal 4 aktivieren / Enable grinding signal 4 / Habilitar señal de rectificado 4
      A_InKeyGEn5 : Bool;   // Schleifsignal 5 aktivieren / Enable grinding signal 5 / Habilitar señal de rectificado 5
      A_InKeyGEn6 : Bool;   // Schleifsignal 6 aktivieren / Enable grinding signal 6 / Habilitar señal de rectificado 6
      A_InKeyGEn7 : Bool;   // Schleifsignal 7 aktivieren / Enable grinding signal 7 / Habilitar señal de rectificado 7
      A_InKeyGEn8 : Bool;   // Schleifsignal 8 aktivieren / Enable grinding signal 8 / Habilitar señal de rectificado 8
      A_InKeyGRunIn1 : Bool;   // Schleiffunktion 1 durchführen / Run grinding function 1 / Ejecutar función de rectificado 1
      A_InKeyGRunIn2 : Bool;   // Schleiffunktion 2 durchführen / Run grinding function 2 / Ejecutar función de rectificado 2
      A_InKeyGRunIn3 : Bool;   // Schleiffunktion 3 durchführen / Run grinding function 3 / Ejecutar función de rectificado 3
      A_InKeyGRunIn4 : Bool;   // Schleiffunktion 4 durchführen / Run grinding function 4 / Ejecutar función de rectificado 4
      A_InKeyGRunIn5 : Bool;   // Schleiffunktion 5 durchführen / Run grinding function 5 / Ejecutar función de rectificado 5
      A_InKeyGRunIn6 : Bool;   // Schleiffunktion 6 durchführen / Run grinding function 6 / Ejecutar función de rectificado 6
      A_InKeyGRunIn7 : Bool;   // Schleiffunktion 7 durchführen / Run grinding function 7 / Ejecutar función de rectificado 7
      A_InKeyGRunIn8 : Bool;   // Schleiffunktion 8 durchführen / Run grinding function 8 / Ejecutar función de rectificado 8
      E_TransformNo : Byte;   // Nummer der aktiven Transformation / Active transformation number / Número de la transformación activa
      f389 : Byte;
      E_InKeyGIsEn1 : Bool;   // Schleifsignal 1 aktiviert / Grinding signal 1 enabled / Señal de rectificado 1 activada
      E_InKeyGIsEn2 : Bool;   // Schleifsignal 2 aktiviert / Grinding signal 2 enabled / Señal de rectificado 2 activada
      E_InKeyGIsEn3 : Bool;   // Schleifsignal 3 aktiviert / Grinding signal 3 enabled / Señal de rectificado 3 activada
      E_InKeyGIsEn4 : Bool;   // Schleifsignal 4 aktiviert / Grinding signal 4 enabled / Señal de rectificado 4 activada
      E_InKeyGIsEn5 : Bool;   // Schleifsignal 5 aktiviert / Grinding signal 5 enabled / Señal de rectificado 5 activada
      E_InKeyGIsEn6 : Bool;   // Schleifsignal 6 aktiviert / Grinding signal 6 enabled / Señal de rectificado 6 activada
      E_InKeyGIsEn7 : Bool;   // Schleifsignal 7 aktiviert / Grinding signal 7 enabled / Señal de rectificado 7 activada
      E_InKeyGIsEn8 : Bool;   // Schleifsignal 8 aktiviert / Grinding signal 8 enabled / Señal de rectificado 8 activada
      E_InKeyGRunOut1 : Bool;   // NCK-Status von Schleiffunktion 1 / NCK status of grinding function 1 / Estado NCK de función de rectificado 1
      E_InKeyGRunOut2 : Bool;   // NCK-Status von Schleiffunktion 3 / NCK status of grinding function 3 / Estado NCK de función de rectificado 3
      E_InKeyGRunOut3 : Bool;   // NCK-Status von Schleiffunktion 3 / NCK status of grinding function 3 / Estado NCK de función de rectificado 3
      E_InKeyGRunOut4 : Bool;   // NCK-Status von Schleiffunktion 4 / NCK status of grinding function 4 / Estado NCK de función de rectificado 4
      E_InKeyGRunOut5 : Bool;   // NCK-Status von Schleiffunktion 5 / NCK status of grinding function 5 / Estado NCK de función de rectificado 5
      E_InKeyGRunOut6 : Bool;   // NCK-Status von Schleiffunktion 6 / NCK status of grinding function 6 / Estado NCK de función de rectificado 6
      E_InKeyGRunOut7 : Bool;   // NCK-Status von Schleiffunktion 7 / NCK status of grinding function 7 / Estado NCK de función de rectificado 7
      E_InKeyGRunOut8 : Bool;   // NCK-Status von Schleiffunktion 8 / NCK status of grinding function 8 / Estado NCK de función de rectificado 8
      E_CART_JOG_MODE : Byte;   // Koordinatensystem für kartesisches Verfahren im Tippbetrieb / Coordinate system for Cartesian jog traverse / Sistema de coordenadas para desplazamiento cartesiano en JOG
      f393 : Byte;
      f394 : Byte;
      f395 : Byte;
      H1_DInt : DInt;   // H-Funktion 1 (DInt) / H Function 1 (DInt) / Función H 1 (DInt)
      H2_DInt : DInt;   // H-Funktion 2 (DInt) / H Function 2 (DInt) / Función H 2 (DInt)
      H3_DInt : DInt;   // H-Funktion 3 (DInt) / H Function 3 (DInt) / Función H 3 (DInt)
      E_AxisSelType : Byte;   // 0: MaschAchse, 1: GeoAchse / 0: MachAxis, 1: GeoAxis / 0: EjeMáq, 1: EjeGeo
      E_AxisSelAxis : Byte;   // Achsnummer / Axis number / Número de eje
      E_AxisSelRequest : Bool;   // Achsauswahl (Touch) / Axis selection (touch) / Selección de eje (táctil)
      f410_1 : Bool;
      f410_2 : Bool;
      f410_3 : Bool;
      f410_4 : Bool;
      f410_5 : Bool;
      f410_6 : Bool;
      f410_7 : Bool;
      f411 : Byte;
      A_AxisSelTypeActive : Byte;   // 0: MaschAchse, 1: GeoAchse (Rücksprung) / 0: MachAxis, 1: GeoAxis (return) / 0: EjeMáq, 1: EjeGeo (salto atrás)
      A_AxisSelAxisActive : Byte;   // Achsnummer (Rücksprung) / Axis number (return) / Número de eje (salto atrás)
   END_STRUCT;
   // // A_Geo[2].HW1 : Handrad 1 aktivieren / Activate handwheel 1 / Activar volante 1
   // // A_Geo[3].HW1 : Handrad 1 aktivieren / Activate handwheel 1 / Activar volante 1
   // // A_Geo[2].HW2 : Handrad 2 aktivieren / Activate handwheel 2 / Activar volante 2
   // // A_Geo[3].HW2 : Handrad 2 aktivieren / Activate handwheel 2 / Activar volante 2
   // // A_Geo[2].HW3 : Handrad 3 aktivieren / Activate handwheel 3 / Activar volante 3
   // // A_Geo[3].HW3 : Handrad 3 aktivieren / Activate handwheel 3 / Activar volante 3
   // // A_Geo[2].FDStop : Vorschub Stopp / Feedrate stop / Parada de avance
   // // A_Geo[3].FDStop : Vorschub Stopp / Feedrate stop / Parada de avance
   // // A_Geo[2].Disabl : Verfahrtaste deaktivieren / Traversing key disable / Desactivar tecla de desplazamiento
   // // A_Geo[3].Disabl : Verfahrtaste deaktivieren / Traversing key disable / Desactivar tecla de desplazamiento
   // // A_Geo[2].RapidTrOR : Eilgang Override / Rapid traverse override / Corregir rápido
   // // A_Geo[3].RapidTrOR : Eilgang Override / Rapid traverse override / Corregir rápido
   // // A_Geo[2].Minus : Verfahrtaste minus / Traversing key minus / Tecla desplazamiento Menos
   // // A_Geo[3].Minus : Verfahrtaste minus / Traversing key minus / Tecla desplazamiento Menos
   // // A_Geo[2].Plus : Verfahrtaste plus / Traversing key plus / Tecla desplazamiento Más
   // // A_Geo[3].Plus : Verfahrtaste plus / Traversing key plus / Tecla desplazamiento Más
   // // A_Geo[2].INC1 : INC 1
   // // A_Geo[3].INC1 : INC 1
   // // A_Geo[2].INC10 : INC 10
   // // A_Geo[3].INC10 : INC 10
   // // A_Geo[2].INC100 : INC 100
   // // A_Geo[3].INC100 : INC 100
   // // A_Geo[2].INC1000 : INC 1000
   // // A_Geo[3].INC1000 : INC 1000
   // // A_Geo[2].INC10000 : INC 10000
   // // A_Geo[3].INC10000 : INC 10000
   // // A_Geo[2].INCVar : INC-Variable / INC variable / Variable INC
   // // A_Geo[3].INCVar : INC-Variable / INC variable / Variable INC
   // // A_Geo[2].ContManTravel : Kontinuierliches Verfahren von Hand / Continuous manual travel / Desplazamiento continuo a mano
   // // A_Geo[3].ContManTravel : Kontinuierliches Verfahren von Hand / Continuous manual travel / Desplazamiento continuo a mano
   // // A_Geo[2].OEM : OEM-Signale / OEM signals / Señales OEM
   // // A_Geo[3].OEM : OEM-Signale / OEM signals / Señales OEM
   // // A_Geo[2].InvHWDirOfRot : Handrad-Drehrichtung umkehren / Invert handwheel direction of rotation / Invertir sentido de giro de volante
   // // A_Geo[3].InvHWDirOfRot : Handrad-Drehrichtung umkehren / Invert handwheel direction of rotation / Invertir sentido de giro de volante
   // // A_Geo[1] : Steuersignale für Geometrieachse [1..3] / Control signals for geometry axis [1..3] / Señales de control para eje geométrico [1..3]
   // // A_Geo[2] : Steuersignale für Geometrieachse [1..3] / Control signals for geometry axis [1..3] / Señales de control para eje geométrico [1..3]
   // // A_Geo[3] : Steuersignale für Geometrieachse [1..3] / Control signals for geometry axis [1..3] / Señales de control para eje geométrico [1..3]
   // // E_Geo[2].HW1 : Handrad 1 aktiv / Handwheel 1 active / Volante 1 activo
   // // E_Geo[3].HW1 : Handrad 1 aktiv / Handwheel 1 active / Volante 1 activo
   // // E_Geo[2].HW2 : Handrad 2 aktiv / Handwheel 2 active / Volante 2 activo
   // // E_Geo[3].HW2 : Handrad 2 aktiv / Handwheel 2 active / Volante 2 activo
   // // E_Geo[2].HW3 : Handrad 3 aktiv / Handwheel 3 active / Volante 3 activo
   // // E_Geo[3].HW3 : Handrad 3 aktiv / Handwheel 3 active / Volante 3 activo
   // // E_Geo[2].TReqMinus : Verfahranforderungen minus / Travel requests minus / Solicitudes de desplazamiento Menos
   // // E_Geo[3].TReqMinus : Verfahranforderungen minus / Travel requests minus / Solicitudes de desplazamiento Menos
   // // E_Geo[2].TReqPlus : Verfahranforderungen plus / Travel requests plus / Solicitudes de desplazamiento Más
   // // E_Geo[3].TReqPlus : Verfahranforderungen plus / Travel requests plus / Solicitudes de desplazamiento Más
   // // E_Geo[2].TCMinus : Verfahrbefehl minus / Traverse command minus / Comando de desplazamiento Menos
   // // E_Geo[3].TCMinus : Verfahrbefehl minus / Traverse command minus / Comando de desplazamiento Menos
   // // E_Geo[2].TCPlus : Verfahrbefehl plus / Traverse command plus / Comando de desplazamiento Más
   // // E_Geo[3].TCPlus : Verfahrbefehl plus / Traverse command plus / Comando de desplazamiento Más
   // // E_Geo[2].INC1 : INC 1 aktiv / INC 1 active / INC 1 activo
   // // E_Geo[3].INC1 : INC 1 aktiv / INC 1 active / INC 1 activo
   // // E_Geo[2].INC10 : INC 10 aktiv / INC 10 active / INC 10 activo
   // // E_Geo[3].INC10 : INC 10 aktiv / INC 10 active / INC 10 activo
   // // E_Geo[2].INC100 : INC 100 aktiv / INC 100 active / INC 100 activo
   // // E_Geo[3].INC100 : INC 100 aktiv / INC 100 active / INC 100 activo
   // // E_Geo[2].INC1000 : INC 1000 aktiv / INC 1000 active / INC 1000 activo
   // // E_Geo[3].INC1000 : INC 1000 aktiv / INC 1000 active / INC 1000 activo
   // // E_Geo[2].INC10000 : INC 10000 aktiv / INC 10000 active / INC 10000 activo
   // // E_Geo[3].INC10000 : INC 10000 aktiv / INC 10000 active / INC 10000 activo
   // // E_Geo[2].INCVar : INC-Variable aktiv / INC variable active / Variable INC activa
   // // E_Geo[3].INCVar : INC-Variable aktiv / INC variable active / Variable INC activa
   // E_Geo[1].ContManTravelAct := false;
   // // E_Geo[2].ContManTravelAct : Kontinuierliches manuelles Verfahren aktiv / Continuous manual travel active / Desplazamiento manual continuo activo
   // // E_Geo[3].ContManTravelAct : Kontinuierliches manuelles Verfahren aktiv / Continuous manual travel active / Desplazamiento manual continuo activo
   // E_Geo[1].f1_7 := false;
   // // E_Geo[2].OEM : OEM-Signale / OEM signals / Señales OEM
   // // E_Geo[3].OEM : OEM-Signale / OEM signals / Señales OEM
   // // E_Geo[2].InvHWDirOfRot : Handrad-Drehrichtung invertiert aktiv / Handwheel direction of rotation invert actively / Invertir activamente sentido de giro volante
   // // E_Geo[3].InvHWDirOfRot : Handrad-Drehrichtung invertiert aktiv / Handwheel direction of rotation invert actively / Invertir activamente sentido de giro volante
   // // E_Geo[1] : Statussignale der Geometrieachse [1..3] / Status signals of geometry axis [1..3] / Señales de estado del eje geométrico [1..3]
   // // E_Geo[2] : Statussignale der Geometrieachse [1..3] / Status signals of geometry axis [1..3] / Señales de estado del eje geométrico [1..3]
   // // E_Geo[3] : Statussignale der Geometrieachse [1..3] / Status signals of geometry axis [1..3] / Señales de estado del eje geométrico [1..3]
   // // A_Ori[2].HW1 : Handrad 1 aktivieren / Activate handwheel 1 / Activar volante 1
   // // A_Ori[3].HW1 : Handrad 1 aktivieren / Activate handwheel 1 / Activar volante 1
   // // A_Ori[2].HW2 : Handrad 2 aktivieren / Activate handwheel 2 / Activar volante 2
   // // A_Ori[3].HW2 : Handrad 2 aktivieren / Activate handwheel 2 / Activar volante 2
   // // A_Ori[2].HW3 : Handrad 3 aktivieren / Activate handwheel 3 / Activar volante 3
   // // A_Ori[3].HW3 : Handrad 3 aktivieren / Activate handwheel 3 / Activar volante 3
   // // A_Ori[2].FDStop : Vorschub Stopp / Feedrate stop / Parada de avance
   // // A_Ori[3].FDStop : Vorschub Stopp / Feedrate stop / Parada de avance
   // // A_Ori[2].Disabl : Verfahrtaste sperren / Traversing key lock / Bloquear tecla desplazamiento
   // // A_Ori[3].Disabl : Verfahrtaste sperren / Traversing key lock / Bloquear tecla desplazamiento
   // // A_Ori[2].RapidTrOR : Eilgang Override / Rapid traverse override / Corregir rápido
   // // A_Ori[3].RapidTrOR : Eilgang Override / Rapid traverse override / Corregir rápido
   // // A_Ori[2].Minus : Verfahrtaste minus / Traversing key minus / Tecla desplazamiento Menos
   // // A_Ori[3].Minus : Verfahrtaste minus / Traversing key minus / Tecla desplazamiento Menos
   // // A_Ori[2].Plus : Verfahrtaste plus / Traversing key plus / Tecla desplazamiento Más
   // // A_Ori[3].Plus : Verfahrtaste plus / Traversing key plus / Tecla desplazamiento Más
   // // A_Ori[2].INC1 : INC 1 aktiv / INC 1 active / INC 1 activo
   // // A_Ori[3].INC1 : INC 1 aktiv / INC 1 active / INC 1 activo
   // // A_Ori[2].INC10 : INC 10 aktiv / INC 10 active / INC 10 activo
   // // A_Ori[3].INC10 : INC 10 aktiv / INC 10 active / INC 10 activo
   // // A_Ori[2].INC100 : INC 100 aktiv / INC 100 active / INC 100 activo
   // // A_Ori[3].INC100 : INC 100 aktiv / INC 100 active / INC 100 activo
   // // A_Ori[2].INC1000 : INC 1000 aktiv / INC 1000 active / INC 1000 activo
   // // A_Ori[3].INC1000 : INC 1000 aktiv / INC 1000 active / INC 1000 activo
   // // A_Ori[2].INC10000 : INC 10000 aktiv / INC 10000 active / INC 10000 activo
   // // A_Ori[3].INC10000 : INC 10000 aktiv / INC 10000 active / INC 10000 activo
   // // A_Ori[2].INCVar : INC-Variable aktiv / INC variable active / Variable INC activa
   // // A_Ori[3].INCVar : INC-Variable aktiv / INC variable active / Variable INC activa
   // // A_Ori[2].OEM : OEM-Signale / OEM signals / Señales OEM
   // // A_Ori[3].OEM : OEM-Signale / OEM signals / Señales OEM
   // // A_Ori[2].InvHWDirOfRot : Drehrichtung Handrad umkehren / Inverting handwheel direction of rotation / Invertir sentido de giro volante
   // // A_Ori[3].InvHWDirOfRot : Drehrichtung Handrad umkehren / Inverting handwheel direction of rotation / Invertir sentido de giro volante
   // // A_Ori[1] : Steuersignale für Orientierungsachsen [1..3] / Control signals for orientation axes [1..3] / Señales de control para ejes de orientación [1..3]
   // // A_Ori[2] : Steuersignale für Orientierungsachsen [1..3] / Control signals for orientation axes [1..3] / Señales de control para ejes de orientación [1..3]
   // // A_Ori[3] : Steuersignale für Orientierungsachsen [1..3] / Control signals for orientation axes [1..3] / Señales de control para ejes de orientación [1..3]
   // // E_Ori[2].HW1 : Handrad 1 aktiv / Handwheel 1 active / Volante 1 activo
   // // E_Ori[3].HW1 : Handrad 1 aktiv / Handwheel 1 active / Volante 1 activo
   // // E_Ori[2].HW2 : Handrad 2 aktiv / Handwheel 2 active / Volante 2 activo
   // // E_Ori[3].HW2 : Handrad 2 aktiv / Handwheel 2 active / Volante 2 activo
   // // E_Ori[2].HW3 : Handrad 3 aktiv / Handwheel 3 active / Volante 3 activo
   // // E_Ori[3].HW3 : Handrad 3 aktiv / Handwheel 3 active / Volante 3 activo
   // // E_Ori[2].TReqMinus : Verfahranforderungen minus / Travel requests minus / Solicitudes de desplazamiento Menos
   // // E_Ori[3].TReqMinus : Verfahranforderungen minus / Travel requests minus / Solicitudes de desplazamiento Menos
   // // E_Ori[2].TReqPlus : Verfahranforderungen plus / Travel requests plus / Solicitudes de desplazamiento Más
   // // E_Ori[3].TReqPlus : Verfahranforderungen plus / Travel requests plus / Solicitudes de desplazamiento Más
   // // E_Ori[2].TCMinus : Verfahrbefehl minus / Traverse command minus / Comando de desplazamiento Menos
   // // E_Ori[3].TCMinus : Verfahrbefehl minus / Traverse command minus / Comando de desplazamiento Menos
   // // E_Ori[2].TCPlus : Verfahrbefehl plus / Traverse command plus / Comando de desplazamiento Más
   // // E_Ori[3].TCPlus : Verfahrbefehl plus / Traverse command plus / Comando de desplazamiento Más
   // // E_Ori[2].INC1 : INC 1 aktiv / INC 1 active / INC 1 activo
   // // E_Ori[3].INC1 : INC 1 aktiv / INC 1 active / INC 1 activo
   // // E_Ori[2].INC10 : INC 10 aktiv / INC 10 active / INC 10 activo
   // // E_Ori[3].INC10 : INC 10 aktiv / INC 10 active / INC 10 activo
   // // E_Ori[2].INC100 : INC 100 aktiv / INC 100 active / INC 100 activo
   // // E_Ori[3].INC100 : INC 100 aktiv / INC 100 active / INC 100 activo
   // // E_Ori[2].INC1000 : INC 1000 aktiv / INC 1000 active / INC 1000 activo
   // // E_Ori[3].INC1000 : INC 1000 aktiv / INC 1000 active / INC 1000 activo
   // // E_Ori[2].INC10000 : INC 10000 aktiv / INC 10000 active / INC 10000 activo
   // // E_Ori[3].INC10000 : INC 10000 aktiv / INC 10000 active / INC 10000 activo
   // // E_Ori[2].INCVar : INC-Variable aktiv / INC variable active / Variable INC activa
   // // E_Ori[3].INCVar : INC-Variable aktiv / INC variable active / Variable INC activa
   // // E_Ori[2].OEM : OEM-Signale / OEM signals / Señales OEM
   // // E_Ori[3].OEM : OEM-Signale / OEM signals / Señales OEM
   // // E_Ori[2].InvHWDirOfRot : Handrad-Drehrichtung invertiert aktiv / Handwheel direction of rotation invert actively / Invertir activamente sentido de giro volante
   // // E_Ori[3].InvHWDirOfRot : Handrad-Drehrichtung invertiert aktiv / Handwheel direction of rotation invert actively / Invertir activamente sentido de giro volante
   // // E_Ori[1] : Steuersignale für Orientierungsachsen [1..3] / Control signals for orientation axes [1..3] / Señales de control para ejes de orientación [1..3]
   // // E_Ori[2] : Steuersignale für Orientierungsachsen [1..3] / Control signals for orientation axes [1..3] / Señales de control para ejes de orientación [1..3]
   // // E_Ori[3] : Steuersignale für Orientierungsachsen [1..3] / Control signals for orientation axes [1..3] / Señales de control para ejes de orientación [1..3]
END_TYPE
